(* IEC 61131-3 sources: SRCI/RobotLibrary/Library/Functions/Convert/DT, 5 files *)

(* ---- DATE_TO_IEC_DATE.st ---- *)
FUNCTION DATE_TO_IEC_DATE : IEC_DATE
// -------------------------------------------------------------------------
//  SRCI Robot Library
// -------------------------------------------------------------------------
//
//  Object:      DATE_TO_IEC_DATE
//  Author:      Thorsten Brach
//  Date:        2024-06-01
//
//  Description:
//
//
//  Copyright:
//    (C) 2024 Thorsten Brach. All rights reserved
//             Licensed under the LGPL-3.0 license.
//
//  Disclaimer:
//    This project is provided without any guarantee and can be used for
//    private and commercial purposes. Any use is at the user’s
//    own risk and responsibility.
//
// -------------------------------------------------------------------------
VAR_INPUT
  Value    : DATE;
END_VAR

VAR
 _tmpDate1 : DWORD;
 _tmpDate2 : DWORD;
 _initDate : DATE := DATE#1990-01-01;
 END_VAR

  // Siemens Dateformat is Day since 01.01.1990
  // TwinCat Dateformat is seconds sinde 01.01.1970
  // Calculation :
  // ( [TwinCat current date] - [ TwinCat 01.01.1970] ) / [Seconds a Day] = Days sinde 01.01.1990 (Siemens Format)

  // copy date to dword
  SysDepMemCpy( pDest := ADR(_tmpDate1), pSrc := ADR( Value   ), DataLen := SIZEOF( Value   ));
  // copy date to dword
  SysDepMemCpy( pDest := ADR(_tmpDate2), pSrc := ADR(_initDate), DataLen := SIZEOF(_initDate));

  // calculate IEC Date :
  DATE_TO_IEC_DATE := UDINT_TO_UINT((_tmpDate1 - _tmpDate2) / 86400); // 86400 Seconds = 1 day

END_FUNCTION

(* ---- IEC_TIMESTAMP_TO_DT.st ---- *)
FUNCTION IEC_TIMESTAMP_TO_DT : DT
// -------------------------------------------------------------------------
//  SRCI Robot Library
// -------------------------------------------------------------------------
//
//  Object:      TIME_TO_IEC_TIME
//  Author:      Thorsten Brach
//  Date:        2025-01-05
//
//  Description:
//
//
//  Copyright:
//    (C) 2025 Thorsten Brach. All rights reserved
//             Licensed under the LGPL-3.0 license.
//
//  Disclaimer:
//    This project is provided without any guarantee and can be used for
//    private and commercial purposes. Any use is at the user’s
//    own risk and responsibility.
//
// -------------------------------------------------------------------------
VAR_INPUT
  Value : IEC_TIMESTAMP;
END_VAR

VAR
  /// internal date
 _date    : DATE;
  /// internal date as string
 _dateStr : STRING;
  /// internal time
 _time    : TOD;
  /// internal time as string
 _timeStr : STRING;
END_VAR

  _date := IEC_DATE_TO_DATE(Value.IEC_DATE);
  _time := IEC_TIME_TO_TIME(Value.IEC_TIME);

  // Example : DATE#2025-1-5
  _dateStr := DATE_TO_STRING(_date);
  // Example : DT#2025-1-5
  _dateStr := strReplace(_dateStr, 'D#', 'DT#');

  // Example : TOD#15:18:4.567
  _timeStr :=  TOD_TO_STRING(_time);
  // Example : -15:18:4.567
  _timeStr := strReplace(_timeStr, 'TOD#', '-');

  // Example : DT#2025-1-5-15:18:4.567
  IEC_TIMESTAMP_TO_DT := STRING_TO_DT( Concat(_dateStr,_timeStr));

END_FUNCTION

(* ---- IEC_TIMESTAMP_TO_SYSTEMTIME.st ---- *)
FUNCTION IEC_TIMESTAMP_TO_SYSTEMTIME : SystemTime
// -------------------------------------------------------------------------
//  SRCI Robot Library
// -------------------------------------------------------------------------
//
//  Object:      IEC_TIMESTAMP_TO_SYSTEMTIME
//  Author:      Thorsten Brach
//  Date:        2025-01-05
//
//  Description:
//
//
//  Copyright:
//    (C) 2025 Thorsten Brach. All rights reserved
//             Licensed under the LGPL-3.0 license.
//
//  Disclaimer:
//    This project is provided without any guarantee and can be used for
//    private and commercial purposes. Any use is at the user’s
//    own risk and responsibility.
//
// -------------------------------------------------------------------------
VAR_INPUT
  Value : IEC_TIMESTAMP;
END_VAR

VAR
  /// internal date
 _date    : DATE;
  /// internal date as string
 _dateStr : STRING;
  /// internal time
 _time    : TOD;
  /// internal time as string
 _timeStr : STRING;
END_VAR

  IEC_TIMESTAMP_TO_SYSTEMTIME.SystemDate := IEC_DATE_TO_DATE(Value.IEC_DATE);
  IEC_TIMESTAMP_TO_SYSTEMTIME.SystemTime := IEC_TIME_TO_TIME(Value.IEC_TIME);

END_FUNCTION

(* ---- SYSTEMTIME_TO_IEC_TIMESTAMP.st ---- *)
FUNCTION SYSTEMTIME_TO_IEC_TIMESTAMP : IEC_TIMESTAMP
// -------------------------------------------------------------------------
//  SRCI Robot Library
// -------------------------------------------------------------------------
//
//  Object:      SYSTEMTIME_TO_IEC_TIMESTAMP
//  Author:      Thorsten Brach
//  Date:        2025-03-30
//
//  Description:
//
//
//  Copyright:
//    (C) 2025 Thorsten Brach. All rights reserved
//             Licensed under the LGPL-3.0 license.
//
//  Disclaimer:
//    This project is provided without any guarantee and can be used for
//    private and commercial purposes. Any use is at the user’s
//    own risk and responsibility.
//
// -------------------------------------------------------------------------
VAR_INPUT
  SystemTime : SystemTime;
END_VAR

  SYSTEMTIME_TO_IEC_TIMESTAMP.IEC_DATE := DATE_TO_IEC_DATE(SystemTime.SystemDate);
  SYSTEMTIME_TO_IEC_TIMESTAMP.IEC_TIME := TIME_TO_IEC_TIME(SystemTime.SystemTime);

END_FUNCTION

(* ---- TIME_TO_IEC_TIME.st ---- *)
FUNCTION TIME_TO_IEC_TIME : IEC_TIME
// -------------------------------------------------------------------------
//  SRCI Robot Library
// -------------------------------------------------------------------------
//
//  Object:      TIME_TO_IEC_TIME
//  Author:      Thorsten Brach
//  Date:        2024-06-01
//
//  Description:
//
//
//  Copyright:
//    (C) 2024 Thorsten Brach. All rights reserved
//             Licensed under the LGPL-3.0 license.
//
//  Disclaimer:
//    This project is provided without any guarantee and can be used for
//    private and commercial purposes. Any use is at the user’s
//    own risk and responsibility.
//
// -------------------------------------------------------------------------
VAR_INPUT
  Value : TOD;
END_VAR

  TIME_TO_IEC_TIME := Value;

END_FUNCTION
